// TIA Portal V18 export
DATA_BLOCK "P01_Control_DB"   // DB22
// stored: InstanceOfName P01_Control, InstanceOfType FB
"P01_Control"
   // VAR_INPUT
   //    I_Start : Bool;
   //    I_Frequency : Real;
   //    I_Alarm_Confirm : Bool;
   // END_VAR
   // VAR
   //    FB_Always_True : Bool;
   //    P01_Modbus_Com_Instance { S7_SetPoint := 'True'} : "P01_TCP_Com";
   // END_VAR
BEGIN
END_DATA_BLOCK
